(* PLC project v0.6.02_RefactorGateAndTest.project, CODESYS CODESYS V3.5 SP19 Patch 1 *)
(* stored: creationDateTime 2026-08-16T00:42:36.465037, modificationDateTime 2026-08-16T00:42:36.465037 *)

VAR_GLOBAL  (* GVL_Pool - ═══════════════════════════════════════════════════════════════ 💾 GVL_Pool — Pool de ressources CAA File (RSU) ─────────────────────────────────────────────────────────────── 🎯 Rôle : instance globale du pool extender CAA File, pour traiter les jobs async d'écriture fichier (évite ASM_CREATEJOB_FAILED). 📄 Docs : bibliothèque RSU (CAA Resource Management) + CAA File. ═══════════════════════════════════════════════════════════════ *)
  PoolInitDone : BOOL := FALSE;  (* init exécutée une seule fois *)
END_VAR
